FUNCTION_BLOCK FB_GenericLinkedList
VAR_INPUT
END_VAR
VAR_OUTPUT
	bInit : BOOL;
END_VAR
VAR
	
	pHead : POINTER TO ST_LinkedListUnit;
	pTail : POINTER TO ST_LinkedListUnit;
	pPointer : POINTER TO ST_LinkedListUnit; //Helper
	
	//pGetNext : POINTER TO ST_LinkedListUnit;
	nGetNextPosition : UINT := 1;
	
	pGetCurrent : POINTER TO ST_LinkedListUnit;
	nGetCurrentPosition : UINT := 1;
	
	nSizeOfLinkedList : DINT;
	
	bIsEmpty : BOOL := TRUE;
	bIsFull : BOOL;
	nUnitsInTheList : DINT;
	
		//DEBUG:
	//If one of the following variables becomes TRUE, investigation of the cause is mandatory
//--------------------------------------------------------------------------------------------
	bTriedToRelocatePositionZero : BOOL;
//--------------------------------------------------------------------------------------------
END_VAR

METHOD M_AddToHead : BOOL
VAR_INPUT
	pUnitToAdd : POINTER TO ST_LinkedListUnit;
END_VAR
IF bIsFull THEN
	RETURN;
END_IF

IF bIsEmpty THEN
	pHead := pUnitToAdd;
	pGetCurrent := pHead;
	pTail := pHead;
	pPointer := pHead;
ELSE
	pHead^.pPrevious := pUnitToAdd;
	pUnitToAdd^.pNext := pHead;
	pUnitToAdd^.pPrevious := NULL;
	pHead := pUnitToAdd;	
END_IF

nUnitsInTheList := nUnitsInTheList + 1;
M_CheckUnitsInTheList();

M_AddToHead := TRUE;
END_METHOD

METHOD M_AddToTail : BOOL
VAR_INPUT
	pUnitToAdd : POINTER TO ST_LinkedListUnit;
END_VAR
IF bIsFull THEN
	RETURN;
END_IF

IF bIsEmpty THEN
	pHead := pUnitToAdd;
	pGetCurrent := pHead;
	pTail := pHead;
	pPointer := pHead;
ELSE
	pTail^.pNext := pUnitToAdd;
	pUnitToAdd^.pPrevious := pTail;
	pUnitToAdd^.pNext := NULL;
	pTail := pUnitToAdd;	
END_IF

nUnitsInTheList := nUnitsInTheList + 1;
M_CheckUnitsInTheList();
	
M_AddToTail := TRUE;
END_METHOD

METHOD M_CheckUnitsInTheList : BOOL
VAR_INPUT
END_VAR
IF nUnitsInTheList = nSizeOfLinkedList THEN
	bIsFull := TRUE;
ELSIF nUnitsInTheList < nSizeOfLinkedList THEN
	bIsFull := FALSE;
END_IF

IF nUnitsInTheList > 0 THEN
	bIsEmpty := FALSE;
ELSIF nUnitsInTheList = 0 THEN
	bIsEmpty := TRUE;
END_IF
END_METHOD

METHOD M_FindUnit : BOOL
VAR_INPUT
END_VAR
END_METHOD

METHOD M_GetCurrent : POINTER TO ST_LinkedListUnit
VAR_INPUT
END_VAR
IF bIsEmpty THEN
	RETURN;
END_IF

M_GetCurrent := pGetCurrent;
END_METHOD

METHOD M_GetCurrentPosition : UINT
VAR_INPUT
END_VAR
M_GetCurrentPosition := nGetCurrentPosition;
END_METHOD

METHOD M_GetHead : POINTER TO ST_LinkedListUnit
IF bIsEmpty THEN
	RETURN;
END_IF

M_GetHead := pHead;
END_METHOD

//Gets the next Unit and moves the current pointer forward
METHOD M_GetNext : POINTER TO ST_LinkedListUnit
IF bIsEmpty THEN
	RETURN;
END_IF

//If the search pointer reaches the end, reset the counter and the pointer
IF pGetCurrent = NULL THEN
	pGetCurrent := pHead;
	nGetNextPosition := 1;
	M_GetNext := pGetCurrent;
	//pGetCurrent := pGetCurrent^.pNext;
ELSE
	M_GetNext := pGetCurrent;
	//pGetCurrent := pGetCurrent^.pNext;
END_IF
pGetCurrent := pGetCurrent^.pNext;
nGetCurrentPosition := nGetNextPosition;
//IF nGetCurrentPosition = nUnitsInTheList THEN
//	nGetNextPosition := 1;
//ELSE
	nGetNextPosition := nGetNextPosition + 1;
//END_IF
END_METHOD

METHOD M_GetTail : POINTER TO ST_LinkedListUnit
IF bIsEmpty THEN
	RETURN;
END_IF

M_GetTail := pTail;
END_METHOD

METHOD M_InitLinkedList : BOOL
VAR_IN_OUT
    aLinkedListMemory : ARRAY [*] OF ST_LinkedListUnit;
END_VAR
VAR
	i : DINT;
	nLowerBound : DINT;
	nUpperBound : DINT;
END_VAR
IF bInit THEN
	RETURN;
END_IF

nLowerBound := LOWER_BOUND(aLinkedListMemory,1);
nUpperBound := UPPER_BOUND(aLinkedListMemory,1);

nSizeOfLinkedList := (nUpperBound - nLowerBound) + 1;


bIsEmpty := TRUE;
bInit := TRUE;
M_InitLinkedList := TRUE;
END_METHOD

METHOD M_RelocateHeadToTail : BOOL
VAR
	pUnit : POINTER TO ST_LinkedListUnit;
END_VAR
pUnit := M_RemoveAtLocation(1);

IF pUnit = NULL THEN
	RETURN;
END_IF

//If the current element is the head
//reset counters
(*
IF pUnit = pGetCurrent THEN
	pGetCurrent := pGetCurrent^.pNext;
	nGetNextPosition := 2;
	nGetCurrentPosition := 1;
END_IF
*)
IF M_AddToTail(pUnit) THEN
	M_RelocateHeadToTail := TRUE;
END_IF
END_METHOD

METHOD M_RelocateToHead : BOOL
VAR
	pUnit : POINTER TO ST_LinkedListUnit;
END_VAR
pUnit := M_RemoveAtLocation(M_GetCurrentPosition());

IF pUnit = NULL THEN
	RETURN;
END_IF

IF M_AddToHead(pUnit) THEN
	M_RelocateToHead := TRUE;
END_IF
END_METHOD

METHOD M_RelocateToTail : BOOL
VAR_INPUT
END_VAR
VAR
	pUnit : POINTER TO ST_LinkedListUnit;
END_VAR
pUnit := M_RemoveAtLocation(M_GetCurrentPosition());

IF pUnit = NULL THEN
	RETURN;
END_IF

IF M_AddToTail(pUnit) THEN
	M_RelocateToTail := TRUE;
END_IF
END_METHOD

METHOD M_RemoveAtLocation : POINTER TO ST_LinkedListUnit
VAR_INPUT
	in_nLocation : UINT;
END_VAR
VAR
	nCounter : UINT;
END_VAR
IF 	bIsEmpty 
	OR in_nLocation > nUnitsInTheList
	OR in_nLocation = 0
	THEN
	
	IF  in_nLocation = 0 
		AND NOT bIsEmpty 
		THEN
		
		bTriedToRelocatePositionZero := TRUE;
	END_IF
	
	RETURN;
END_IF

pPointer := pHead;
IF in_nLocation = 1 THEN
	M_RemoveAtLocation := M_RemoveHead();
	RETURN;
ELSIF in_nLocation = nUnitsInTheList THEN
	M_RemoveAtLocation := M_RemoveTail();
	RETURN;
ELSE
	
	FOR nCounter := 2 TO in_nLocation DO
		pPointer := pPointer^.pNext;
	END_FOR

END_IF

M_RemoveAtLocation := pPointer;

nUnitsInTheList := nUnitsInTheList - 1;
M_CheckUnitsInTheList();

pPointer := pPointer^.pPrevious;
pPointer^.pNext := pPointer^.pNext^.pNext;
pPointer := pPointer^.pNext;
pPointer^.pPrevious := pPointer^.pPrevious^.pPrevious;
END_METHOD

METHOD M_RemoveHead : POINTER TO ST_LinkedListUnit
VAR_INPUT
END_VAR
IF bIsEmpty THEN
	RETURN;
END_IF

M_RemoveHead := pHead;

IF nUnitsInTheList = 1 THEN
	nUnitsInTheList := 0;
	bIsEmpty := TRUE;	
	pHead := NULL;
	pTail := NULL;
	pPointer := NULL;
ELSE
	pHead := pHead^.pNext;
	pHead^.pPrevious := NULL; 	
	nUnitsInTheList := nUnitsInTheList - 1;
END_IF

M_CheckUnitsInTheList();
END_METHOD

METHOD M_RemoveTail : POINTER TO ST_LinkedListUnit
VAR_INPUT
END_VAR
IF bIsEmpty THEN
	RETURN;
END_IF

M_RemoveTail := pTail;

IF nUnitsInTheList = 1 THEN
	nUnitsInTheList := 0;
	bIsEmpty := TRUE;	
	pHead := NULL;
	pTail := NULL;
	pPointer := NULL;
ELSE
	pTail := pTail^.pPrevious;
	pTail^.pNext := NULL; 	
	nUnitsInTheList := nUnitsInTheList - 1;
END_IF

M_CheckUnitsInTheList();
END_METHOD

END_FUNCTION_BLOCK

(* stored: Version 1.1.0.1, ProductVersion 3.1.4022.16
   POU FB_GenericLinkedList: Id {366e2f0e-7afe-4f4c-97fe-7cd755399221}, SpecialFunc None
   Method M_AddToHead: Id {effdf2ca-9db7-44c2-bac2-468f11eabb39}
   Method M_AddToTail: Id {07db24fe-d9ac-4de5-88fc-850ffc004359}
   Method M_CheckUnitsInTheList: Id {bbd017d8-f695-4908-acb8-669ef5f07432}
   Method M_FindUnit: Id {60e53482-97a0-40ba-bf35-1a1512886224}
   Method M_GetCurrent: Id {27c6129a-a04d-4e80-a1b9-970c50c52625}
   Method M_GetCurrentPosition: Id {05b57a4b-a7d5-456f-8d63-a682ad4188ed}
   Method M_GetHead: Id {3edf442d-b82c-4445-b424-6c63e68bf295}
   Method M_GetNext: Id {a655ed2a-5eac-4ac6-94e0-a8b218a9e90f}
   Method M_GetTail: Id {271d1afe-0efd-48a7-8c68-6f953c85f059}
   Method M_InitLinkedList: Id {113ef8cc-345a-433f-aa32-465314df399e}
   Method M_RelocateHeadToTail: Id {38b8cb2d-facb-4251-97c6-3c7d9b68e457}
   Method M_RelocateToHead: Id {cf6e92ba-f408-4dd7-9d8e-a16459af382f}
   Method M_RelocateToTail: Id {3d3ee349-93fb-412a-b2e0-e553994188ff}
   Method M_RemoveAtLocation: Id {9227fb3e-6a0f-4f71-bd9d-820303e88046}
   Method M_RemoveHead: Id {eeabe269-a852-42ee-a5ca-901cc18c8c4e}
   Method M_RemoveTail: Id {6ac5a376-447f-4738-a4c7-a14fa0bc6d7c} *)
